# EPICS substitutions: db/Beckhoff_1XXX/ecmcEPP1008.substitutions
# generic slave part
file "ecmcEcSlave.template"{
  pattern {}
          {}
}

# binary inputs
file "ecmc_binaryInput-chX.template"{
  pattern {CH_ID}
          {01   }
          {02   }
          {03   }
          {04   }
          {05   }
          {06   }
          {07   }
          {08   }
}
